TYPE ST_StatisticsHMI :
STRUCT
	
	sName					: STRING;
	nGood					: DINT;
	nBad					: DINT;
	bResetGood				: BOOL;
	bResetBad				: BOOL;	
	nEfficency				: STRING;
	
END_STRUCT
END_TYPE

(* stored: Version 1.1.0.1, ProductVersion 3.1.4026.18
   DUT ST_StatisticsHMI: Id {c13f0ccd-71ee-4c5d-9b8e-5212c4fac55e} *)
